Fanuc KAREL source: compact_preamble.KL

PROGRAM KD00003
%CMOSVARS
%NOLOCKGROUP
VAR
I:INTEGER;J:INTEGER;B:BOOLEAN;R:REAL;S : STRING[80]
BEGIN
I=1
END KD00003
